// TIA Portal V17 export
// export: Created 2024-03-30T11:15:12.0014028Z, ExportSetting WithDefaults, DisplayName Totally Integrated Automation Portal, DisplayVersion V17, DisplayName TIA Portal Openness, DisplayVersion V17, DisplayName TIA Portal Version Control Interface, DisplayVersion V17, DisplayName STEP 7 Professional, DisplayVersion V17, DisplayName STEP 7 Safety, DisplayVersion V17, DisplayName WinCC Advanced, DisplayVersion V17
TYPE "typ_VGR_Trigger"
// stored: IsFailsafeCompliant false
   STRUCT
      ldt_ts : LDT;
      i_code : Int;
      Workpiece : "typ_Workpiece";
   END_STRUCT;
END_TYPE
